// TIA Portal V17 export
// export: Created 2025-07-01T09:58:42.1462376Z, ExportSetting WithDefaults, DisplayName Totally Integrated Automation Portal, DisplayVersion V17 Update 8, DisplayName TIA Portal Openness, DisplayVersion V17 Update 8, DisplayName TIA Portal Version Control Interface, DisplayVersion V17, DisplayName SINAMICS Startdrive Advanced, DisplayVersion V17 SP2, DisplayName SINAMICS Startdrive G110M, G120, G120C, G120D, G120P, G115D, DisplayVersion V17 SP2, DisplayName SINAMICS Startdrive G130, G150, S120, S150, SINAMICS MV, S210, DisplayVersion V17 SP2, DisplayName STEP 7 Professional, DisplayVersion V17 Update 8, DisplayName SINUMERIK ONE STEP 7 Toolbox, DisplayVersion V17 Update 12, DisplayName SINUMERIK ONE PLC Basic Program Plus, DisplayVersion V17 Update 12, DisplayName SINUMERIK 840D sl STEP 7 Toolbox, DisplayVersion V17 Update 12, DisplayName STEP 7 Safety, DisplayVersion V17 Update 6, DisplayName WinCC Advanced, DisplayVersion V17 Update 8
FUNCTION "FC2034_DRY_CYCLE" : Void   // FC2034, LAD
{ S7_Optimized_Access := 'FALSE' }
AUTHOR : ETXETAR
VERSION : 1.0
// stored: AutoNumber false, IsIECCheckEnabled false, SetENOAutomatically false, UDAEnableTagReadback false
   VAR_TEMP
      O_BYTE_0 : Struct   // OPTIONS BYTE 0
         MANUAL_LOAD_WITH_LIFT : Bool;   // MANUAL LOAD WITH LIFTING DEVICE OPTION
      END_STRUCT;
      DISABLE_COMMAND : Bool;   // DRY CYCLE DISABLE COMMAND
   END_VAR
   VAR CONSTANT
      FC_NUMBER : DInt := 2034;
   END_VAR
   VAR_TEMP   // added for the SCL form of the ladder/FBD networks
      _w1 : Bool;
      _w2 : Bool;
   END_VAR
BEGIN

REGION Network 1: MANUAL LOAD WITH LIFTING DEVICE OPTION
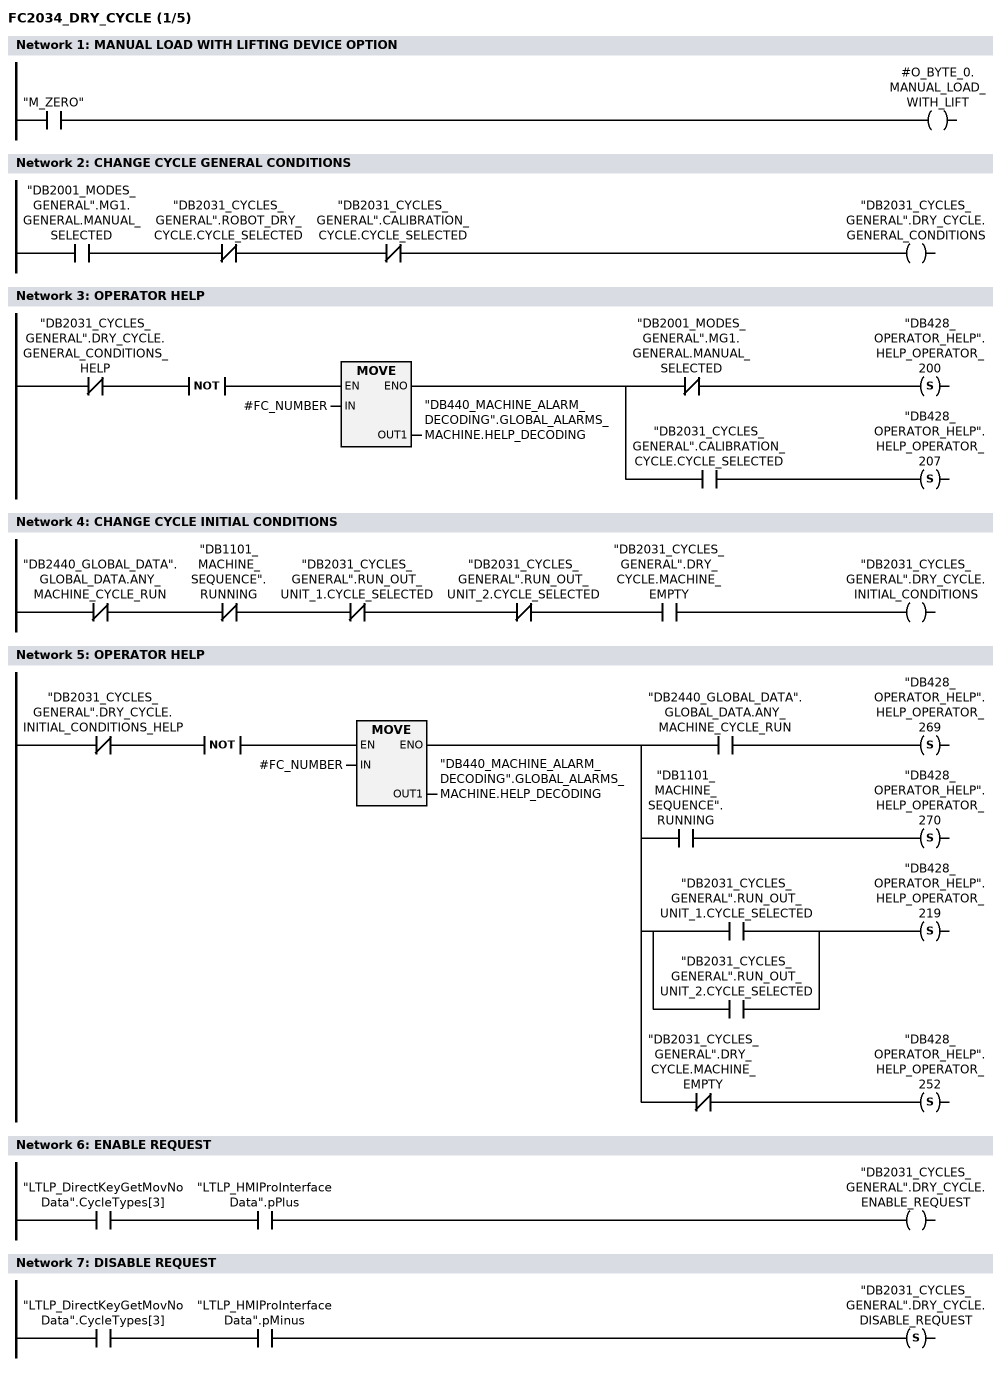
   RUNG wire#powerrail
      Contact( "M_ZERO" )
      Coil( #O_BYTE_0.MANUAL_LOAD_WITH_LIFT )
   END_RUNG
   // the same network as SCL:
   #O_BYTE_0.MANUAL_LOAD_WITH_LIFT := "M_ZERO";
END_REGION

REGION Network 2: CHANGE CYCLE GENERAL CONDITIONS
   RUNG wire#powerrail
      Contact( "DB2001_MODES_GENERAL".MG1.GENERAL.MANUAL_SELECTED )
      I_Contact( "DB2031_CYCLES_GENERAL".ROBOT_DRY_CYCLE.CYCLE_SELECTED )
      I_Contact( "DB2031_CYCLES_GENERAL".CALIBRATION_CYCLE.CYCLE_SELECTED )
      Coil( "DB2031_CYCLES_GENERAL".DRY_CYCLE.GENERAL_CONDITIONS )
   END_RUNG
   // the same network as SCL:
   "DB2031_CYCLES_GENERAL".DRY_CYCLE.GENERAL_CONDITIONS := "DB2001_MODES_GENERAL".MG1.GENERAL.MANUAL_SELECTED AND NOT "DB2031_CYCLES_GENERAL".ROBOT_DRY_CYCLE.CYCLE_SELECTED AND NOT "DB2031_CYCLES_GENERAL".CALIBRATION_CYCLE.CYCLE_SELECTED;
END_REGION

REGION Network 3: OPERATOR HELP
   RUNG wire#powerrail
      I_Contact( "DB2031_CYCLES_GENERAL".DRY_CYCLE.GENERAL_CONDITIONS_HELP )
      Not()
      { S7_GenerateENO := "TRUE" } Move(in := #FC_NUMBER, out1 => "DB440_MACHINE_ALARM_DECODING".GLOBAL_ALARMS_MACHINE.HELP_DECODING)
      wire#w1
      I_Contact( "DB2001_MODES_GENERAL".MG1.GENERAL.MANUAL_SELECTED )
      S_Coil( "DB428_OPERATOR_HELP".HELP_OPERATOR_200 )
   END_RUNG
   RUNG wire#w1
      Contact( "DB2031_CYCLES_GENERAL".CALIBRATION_CYCLE.CYCLE_SELECTED )
      S_Coil( "DB428_OPERATOR_HELP".HELP_OPERATOR_207 )
   END_RUNG
   // the same network as SCL:
   // ENO of a box is taken as its EN; it also drops when the box reports an error
   #_w1 := NOT (NOT "DB2031_CYCLES_GENERAL".DRY_CYCLE.GENERAL_CONDITIONS_HELP);
   IF #_w1 THEN "DB440_MACHINE_ALARM_DECODING".GLOBAL_ALARMS_MACHINE.HELP_DECODING := #FC_NUMBER; END_IF;
   IF #_w1 AND NOT "DB2001_MODES_GENERAL".MG1.GENERAL.MANUAL_SELECTED THEN
       "DB428_OPERATOR_HELP".HELP_OPERATOR_200 := TRUE;
   END_IF;
   IF #_w1 AND "DB2031_CYCLES_GENERAL".CALIBRATION_CYCLE.CYCLE_SELECTED THEN
       "DB428_OPERATOR_HELP".HELP_OPERATOR_207 := TRUE;
   END_IF;
END_REGION

REGION Network 4: CHANGE CYCLE INITIAL CONDITIONS
   RUNG wire#powerrail
      I_Contact( "DB2440_GLOBAL_DATA".GLOBAL_DATA.ANY_MACHINE_CYCLE_RUN )
      I_Contact( "DB1101_MACHINE_SEQUENCE".RUNNING )
      I_Contact( "DB2031_CYCLES_GENERAL".RUN_OUT_UNIT_1.CYCLE_SELECTED )
      I_Contact( "DB2031_CYCLES_GENERAL".RUN_OUT_UNIT_2.CYCLE_SELECTED )
      Contact( "DB2031_CYCLES_GENERAL".DRY_CYCLE.MACHINE_EMPTY )
      Coil( "DB2031_CYCLES_GENERAL".DRY_CYCLE.INITIAL_CONDITIONS )
   END_RUNG
   // the same network as SCL:
   "DB2031_CYCLES_GENERAL".DRY_CYCLE.INITIAL_CONDITIONS := NOT "DB2440_GLOBAL_DATA".GLOBAL_DATA.ANY_MACHINE_CYCLE_RUN AND NOT "DB1101_MACHINE_SEQUENCE".RUNNING AND NOT "DB2031_CYCLES_GENERAL".RUN_OUT_UNIT_1.CYCLE_SELECTED AND NOT "DB2031_CYCLES_GENERAL".RUN_OUT_UNIT_2.CYCLE_SELECTED AND "DB2031_CYCLES_GENERAL".DRY_CYCLE.MACHINE_EMPTY;
END_REGION

REGION Network 5: OPERATOR HELP
   RUNG wire#powerrail
      I_Contact( "DB2031_CYCLES_GENERAL".DRY_CYCLE.INITIAL_CONDITIONS_HELP )
      Not()
      { S7_GenerateENO := "TRUE" } Move(in := #FC_NUMBER, out1 => "DB440_MACHINE_ALARM_DECODING".GLOBAL_ALARMS_MACHINE.HELP_DECODING)
      wire#w1
      Contact( "DB2440_GLOBAL_DATA".GLOBAL_DATA.ANY_MACHINE_CYCLE_RUN )
      S_Coil( "DB428_OPERATOR_HELP".HELP_OPERATOR_269 )
   END_RUNG
   RUNG wire#w1
      Contact( "DB1101_MACHINE_SEQUENCE".RUNNING )
      S_Coil( "DB428_OPERATOR_HELP".HELP_OPERATOR_270 )
   END_RUNG
   RUNG wire#w1
      Contact( "DB2031_CYCLES_GENERAL".RUN_OUT_UNIT_1.CYCLE_SELECTED )
      wire#w2
      S_Coil( "DB428_OPERATOR_HELP".HELP_OPERATOR_219 )
   END_RUNG
   RUNG wire#w1
      Contact( "DB2031_CYCLES_GENERAL".RUN_OUT_UNIT_2.CYCLE_SELECTED )
   END_RUNG wire#w2
   RUNG wire#w1
      I_Contact( "DB2031_CYCLES_GENERAL".DRY_CYCLE.MACHINE_EMPTY )
      S_Coil( "DB428_OPERATOR_HELP".HELP_OPERATOR_252 )
   END_RUNG
   // the same network as SCL:
   // ENO of a box is taken as its EN; it also drops when the box reports an error
   #_w1 := NOT (NOT "DB2031_CYCLES_GENERAL".DRY_CYCLE.INITIAL_CONDITIONS_HELP);
   IF #_w1 THEN "DB440_MACHINE_ALARM_DECODING".GLOBAL_ALARMS_MACHINE.HELP_DECODING := #FC_NUMBER; END_IF;
   IF #_w1 AND "DB2440_GLOBAL_DATA".GLOBAL_DATA.ANY_MACHINE_CYCLE_RUN THEN
       "DB428_OPERATOR_HELP".HELP_OPERATOR_269 := TRUE;
   END_IF;
   IF #_w1 AND "DB1101_MACHINE_SEQUENCE".RUNNING THEN
       "DB428_OPERATOR_HELP".HELP_OPERATOR_270 := TRUE;
   END_IF;
   IF #_w1 AND ("DB2031_CYCLES_GENERAL".RUN_OUT_UNIT_1.CYCLE_SELECTED OR "DB2031_CYCLES_GENERAL".RUN_OUT_UNIT_2.CYCLE_SELECTED) THEN
       "DB428_OPERATOR_HELP".HELP_OPERATOR_219 := TRUE;
   END_IF;
   IF #_w1 AND NOT "DB2031_CYCLES_GENERAL".DRY_CYCLE.MACHINE_EMPTY THEN
       "DB428_OPERATOR_HELP".HELP_OPERATOR_252 := TRUE;
   END_IF;
END_REGION

REGION Network 6: ENABLE REQUEST
   RUNG wire#powerrail
      Contact( "LTLP_DirectKeyGetMovNoData".CycleTypes[3] )
      Contact( "LTLP_HMIProInterfaceData".pPlus )
      Coil( "DB2031_CYCLES_GENERAL".DRY_CYCLE.ENABLE_REQUEST )
   END_RUNG
   // the same network as SCL:
   "DB2031_CYCLES_GENERAL".DRY_CYCLE.ENABLE_REQUEST := "LTLP_DirectKeyGetMovNoData".CycleTypes[3] AND "LTLP_HMIProInterfaceData".pPlus;
END_REGION

REGION Network 7: DISABLE REQUEST
   RUNG wire#powerrail
      Contact( "LTLP_DirectKeyGetMovNoData".CycleTypes[3] )
      Contact( "LTLP_HMIProInterfaceData".pMinus )
      S_Coil( "DB2031_CYCLES_GENERAL".DRY_CYCLE.DISABLE_REQUEST )
   END_RUNG
   // the same network as SCL:
   IF "LTLP_DirectKeyGetMovNoData".CycleTypes[3] AND "LTLP_HMIProInterfaceData".pMinus THEN
       "DB2031_CYCLES_GENERAL".DRY_CYCLE.DISABLE_REQUEST := TRUE;
   END_IF;
END_REGION

REGION Network 8: ROBOT DRY CYCLE DISABLE COMMAND
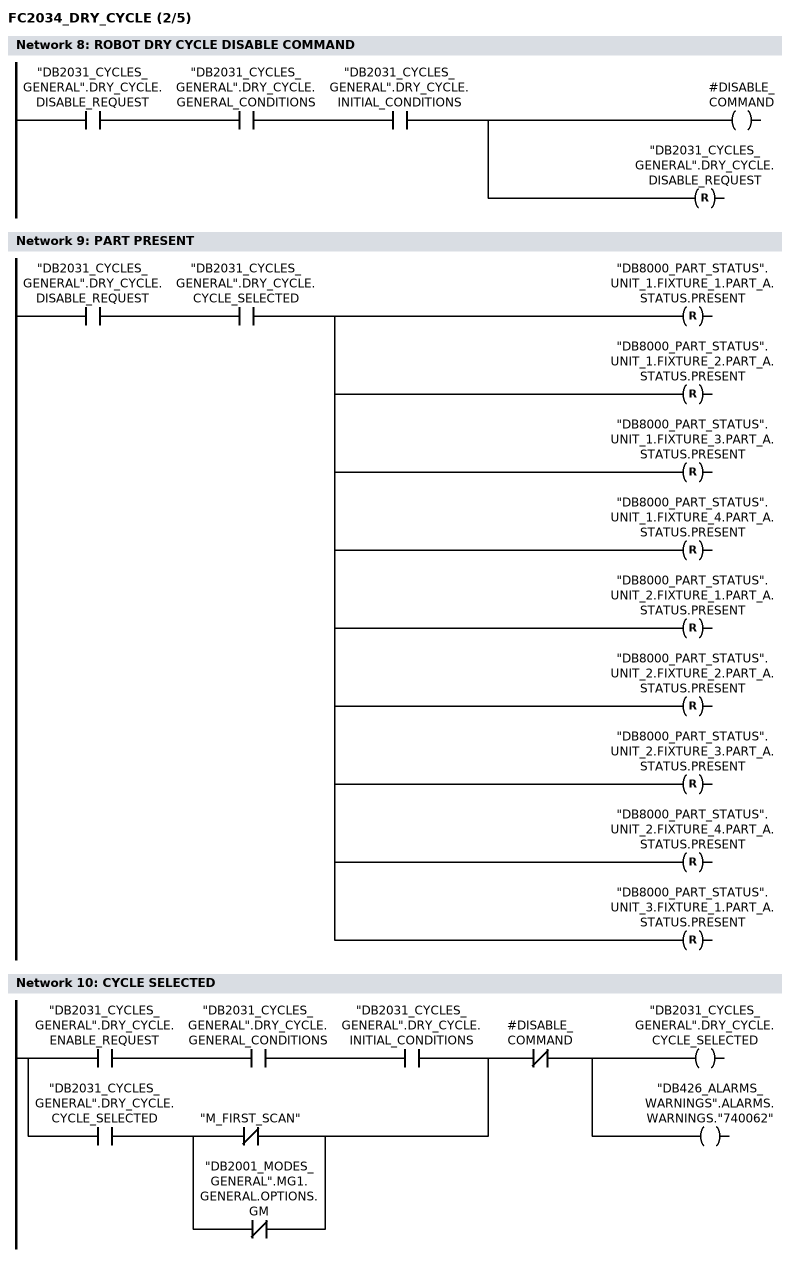
   RUNG wire#powerrail
      Contact( "DB2031_CYCLES_GENERAL".DRY_CYCLE.DISABLE_REQUEST )
      Contact( "DB2031_CYCLES_GENERAL".DRY_CYCLE.GENERAL_CONDITIONS )
      Contact( "DB2031_CYCLES_GENERAL".DRY_CYCLE.INITIAL_CONDITIONS )
      wire#w1
      Coil( #DISABLE_COMMAND )
   END_RUNG
   RUNG wire#w1
      R_Coil( "DB2031_CYCLES_GENERAL".DRY_CYCLE.DISABLE_REQUEST )
   END_RUNG
   // the same network as SCL:
   #DISABLE_COMMAND := "DB2031_CYCLES_GENERAL".DRY_CYCLE.DISABLE_REQUEST AND "DB2031_CYCLES_GENERAL".DRY_CYCLE.GENERAL_CONDITIONS AND "DB2031_CYCLES_GENERAL".DRY_CYCLE.INITIAL_CONDITIONS;
   IF #DISABLE_COMMAND THEN "DB2031_CYCLES_GENERAL".DRY_CYCLE.DISABLE_REQUEST := FALSE; END_IF;
END_REGION

REGION Network 9: PART PRESENT
   RUNG wire#powerrail
      Contact( "DB2031_CYCLES_GENERAL".DRY_CYCLE.DISABLE_REQUEST )
      Contact( "DB2031_CYCLES_GENERAL".DRY_CYCLE.CYCLE_SELECTED )
      wire#w1
      R_Coil( "DB8000_PART_STATUS".UNIT_1.FIXTURE_1.PART_A.STATUS.PRESENT )
   END_RUNG
   RUNG wire#w1
      R_Coil( "DB8000_PART_STATUS".UNIT_1.FIXTURE_2.PART_A.STATUS.PRESENT )
   END_RUNG
   RUNG wire#w1
      R_Coil( "DB8000_PART_STATUS".UNIT_1.FIXTURE_3.PART_A.STATUS.PRESENT )
   END_RUNG
   RUNG wire#w1
      R_Coil( "DB8000_PART_STATUS".UNIT_1.FIXTURE_4.PART_A.STATUS.PRESENT )
   END_RUNG
   RUNG wire#w1
      R_Coil( "DB8000_PART_STATUS".UNIT_2.FIXTURE_1.PART_A.STATUS.PRESENT )
   END_RUNG
   RUNG wire#w1
      R_Coil( "DB8000_PART_STATUS".UNIT_2.FIXTURE_2.PART_A.STATUS.PRESENT )
   END_RUNG
   RUNG wire#w1
      R_Coil( "DB8000_PART_STATUS".UNIT_2.FIXTURE_3.PART_A.STATUS.PRESENT )
   END_RUNG
   RUNG wire#w1
      R_Coil( "DB8000_PART_STATUS".UNIT_2.FIXTURE_4.PART_A.STATUS.PRESENT )
   END_RUNG
   RUNG wire#w1
      R_Coil( "DB8000_PART_STATUS".UNIT_3.FIXTURE_1.PART_A.STATUS.PRESENT )
   END_RUNG
   // the same network as SCL:
   IF "DB2031_CYCLES_GENERAL".DRY_CYCLE.DISABLE_REQUEST AND "DB2031_CYCLES_GENERAL".DRY_CYCLE.CYCLE_SELECTED THEN
       "DB8000_PART_STATUS".UNIT_1.FIXTURE_1.PART_A.STATUS.PRESENT := FALSE;
       "DB8000_PART_STATUS".UNIT_1.FIXTURE_2.PART_A.STATUS.PRESENT := FALSE;
       "DB8000_PART_STATUS".UNIT_1.FIXTURE_3.PART_A.STATUS.PRESENT := FALSE;
       "DB8000_PART_STATUS".UNIT_1.FIXTURE_4.PART_A.STATUS.PRESENT := FALSE;
       "DB8000_PART_STATUS".UNIT_2.FIXTURE_1.PART_A.STATUS.PRESENT := FALSE;
       "DB8000_PART_STATUS".UNIT_2.FIXTURE_2.PART_A.STATUS.PRESENT := FALSE;
       "DB8000_PART_STATUS".UNIT_2.FIXTURE_3.PART_A.STATUS.PRESENT := FALSE;
       "DB8000_PART_STATUS".UNIT_2.FIXTURE_4.PART_A.STATUS.PRESENT := FALSE;
       "DB8000_PART_STATUS".UNIT_3.FIXTURE_1.PART_A.STATUS.PRESENT := FALSE;
   END_IF;
END_REGION

REGION Network 10: CYCLE SELECTED
   RUNG wire#powerrail
      Contact( "DB2031_CYCLES_GENERAL".DRY_CYCLE.ENABLE_REQUEST )
      Contact( "DB2031_CYCLES_GENERAL".DRY_CYCLE.GENERAL_CONDITIONS )
      Contact( "DB2031_CYCLES_GENERAL".DRY_CYCLE.INITIAL_CONDITIONS )
      wire#w1
      I_Contact( #DISABLE_COMMAND )
      wire#w3
      Coil( "DB2031_CYCLES_GENERAL".DRY_CYCLE.CYCLE_SELECTED )
   END_RUNG
   RUNG wire#powerrail
      Contact( "DB2031_CYCLES_GENERAL".DRY_CYCLE.CYCLE_SELECTED )
      wire#w2
      I_Contact( "M_FIRST_SCAN" )
   END_RUNG wire#w1
   RUNG wire#w2
      I_Contact( "DB2001_MODES_GENERAL".MG1.GENERAL.OPTIONS.GM )
   END_RUNG wire#w1
   RUNG wire#w3
      Coil( "DB426_ALARMS_WARNINGS".ALARMS.WARNINGS."740062" )
   END_RUNG
   // the same network as SCL:
   "DB2031_CYCLES_GENERAL".DRY_CYCLE.CYCLE_SELECTED := (("DB2031_CYCLES_GENERAL".DRY_CYCLE.ENABLE_REQUEST AND "DB2031_CYCLES_GENERAL".DRY_CYCLE.GENERAL_CONDITIONS AND "DB2031_CYCLES_GENERAL".DRY_CYCLE.INITIAL_CONDITIONS) OR ("DB2031_CYCLES_GENERAL".DRY_CYCLE.CYCLE_SELECTED AND (NOT "M_FIRST_SCAN" OR NOT "DB2001_MODES_GENERAL".MG1.GENERAL.OPTIONS.GM))) AND NOT #DISABLE_COMMAND;
   "DB426_ALARMS_WARNINGS".ALARMS.WARNINGS."740062" := "DB2031_CYCLES_GENERAL".DRY_CYCLE.CYCLE_SELECTED;
END_REGION

REGION Network 11: WARNINGS
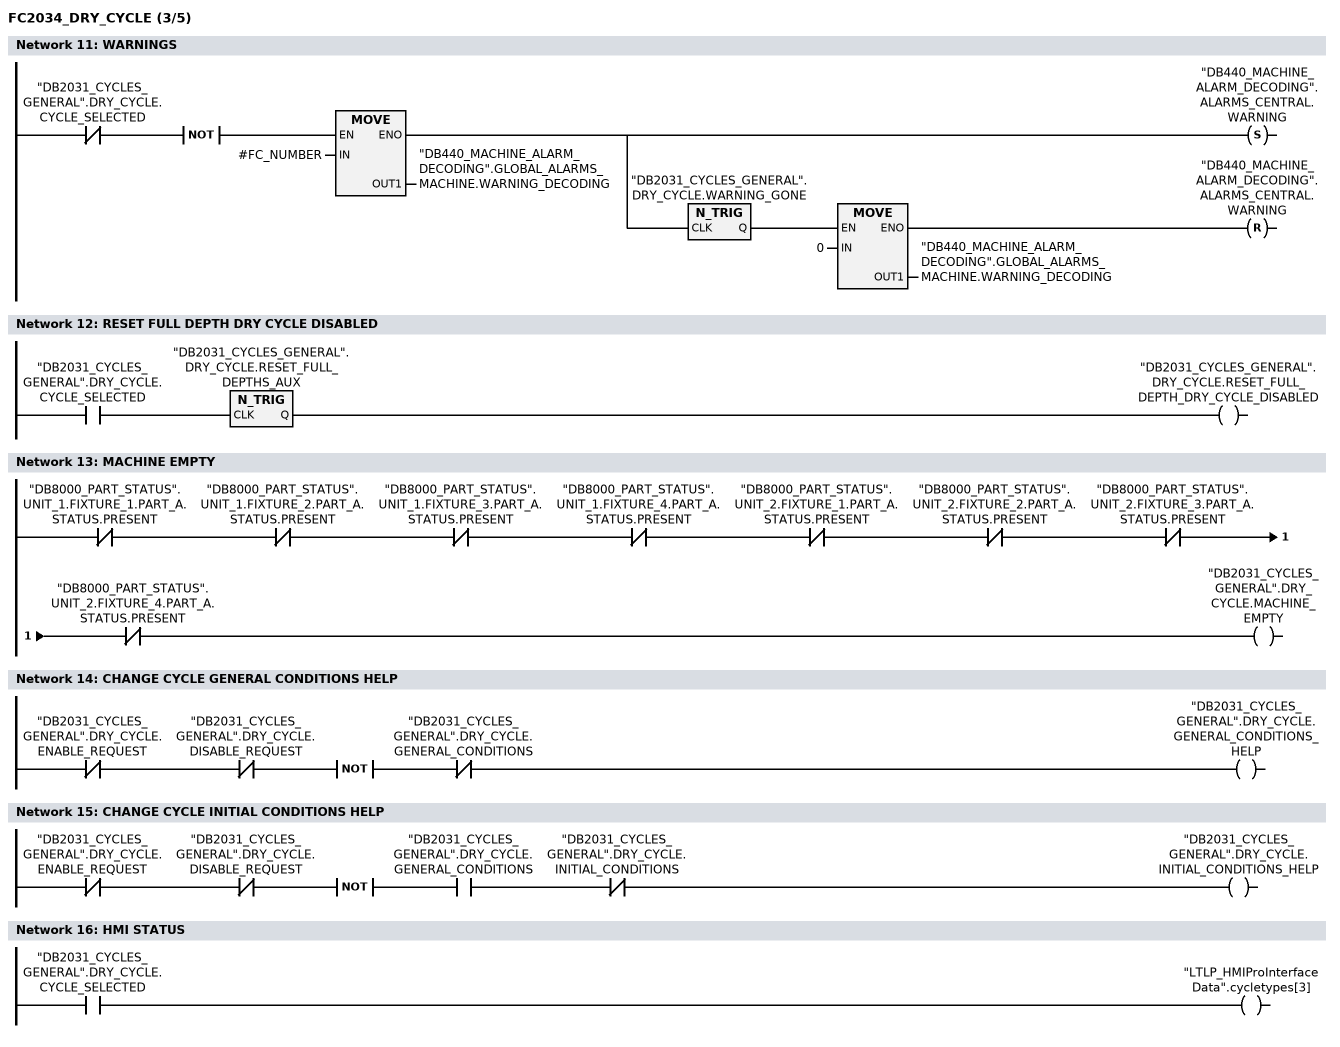
   RUNG wire#powerrail
      I_Contact( "DB2031_CYCLES_GENERAL".DRY_CYCLE.CYCLE_SELECTED )
      Not()
      Move(in := #FC_NUMBER, out1 => "DB440_MACHINE_ALARM_DECODING".GLOBAL_ALARMS_MACHINE.WARNING_DECODING)
      wire#w1
      S_Coil( "DB440_MACHINE_ALARM_DECODING".ALARMS_CENTRAL.WARNING )
   END_RUNG
   RUNG wire#w1
      N_Trig( "DB2031_CYCLES_GENERAL".DRY_CYCLE.WARNING_GONE )
      Move(in := 0, out1 => "DB440_MACHINE_ALARM_DECODING".GLOBAL_ALARMS_MACHINE.WARNING_DECODING)
      R_Coil( "DB440_MACHINE_ALARM_DECODING".ALARMS_CENTRAL.WARNING )
   END_RUNG
   // the same network as SCL:
   #_w1 := NOT (NOT "DB2031_CYCLES_GENERAL".DRY_CYCLE.CYCLE_SELECTED);
   IF #_w1 THEN
       "DB440_MACHINE_ALARM_DECODING".GLOBAL_ALARMS_MACHINE.WARNING_DECODING := #FC_NUMBER;
       "DB440_MACHINE_ALARM_DECODING".ALARMS_CENTRAL.WARNING := TRUE;
   END_IF;
   #_w2 := NOT #_w1 AND "DB2031_CYCLES_GENERAL".DRY_CYCLE.WARNING_GONE;   // falling edge
   "DB2031_CYCLES_GENERAL".DRY_CYCLE.WARNING_GONE := #_w1;
   IF #_w2 THEN
       "DB440_MACHINE_ALARM_DECODING".GLOBAL_ALARMS_MACHINE.WARNING_DECODING := 0;
       "DB440_MACHINE_ALARM_DECODING".ALARMS_CENTRAL.WARNING := FALSE;
   END_IF;
END_REGION

REGION Network 12: RESET FULL DEPTH DRY CYCLE DISABLED
   RUNG wire#powerrail
      Contact( "DB2031_CYCLES_GENERAL".DRY_CYCLE.CYCLE_SELECTED )
      N_Trig( "DB2031_CYCLES_GENERAL".DRY_CYCLE.RESET_FULL_DEPTHS_AUX )
      Coil( "DB2031_CYCLES_GENERAL".DRY_CYCLE.RESET_FULL_DEPTH_DRY_CYCLE_DISABLED )
   END_RUNG
   // the same network as SCL:
   #_w1 := NOT "DB2031_CYCLES_GENERAL".DRY_CYCLE.CYCLE_SELECTED AND "DB2031_CYCLES_GENERAL".DRY_CYCLE.RESET_FULL_DEPTHS_AUX;   // falling edge
   "DB2031_CYCLES_GENERAL".DRY_CYCLE.RESET_FULL_DEPTHS_AUX := "DB2031_CYCLES_GENERAL".DRY_CYCLE.CYCLE_SELECTED;
   "DB2031_CYCLES_GENERAL".DRY_CYCLE.RESET_FULL_DEPTH_DRY_CYCLE_DISABLED := #_w1;
END_REGION

REGION Network 13: MACHINE EMPTY
   RUNG wire#powerrail
      I_Contact( "DB8000_PART_STATUS".UNIT_1.FIXTURE_1.PART_A.STATUS.PRESENT )
      I_Contact( "DB8000_PART_STATUS".UNIT_1.FIXTURE_2.PART_A.STATUS.PRESENT )
      I_Contact( "DB8000_PART_STATUS".UNIT_1.FIXTURE_3.PART_A.STATUS.PRESENT )
      I_Contact( "DB8000_PART_STATUS".UNIT_1.FIXTURE_4.PART_A.STATUS.PRESENT )
      I_Contact( "DB8000_PART_STATUS".UNIT_2.FIXTURE_1.PART_A.STATUS.PRESENT )
      I_Contact( "DB8000_PART_STATUS".UNIT_2.FIXTURE_2.PART_A.STATUS.PRESENT )
      I_Contact( "DB8000_PART_STATUS".UNIT_2.FIXTURE_3.PART_A.STATUS.PRESENT )
      I_Contact( "DB8000_PART_STATUS".UNIT_2.FIXTURE_4.PART_A.STATUS.PRESENT )
      Coil( "DB2031_CYCLES_GENERAL".DRY_CYCLE.MACHINE_EMPTY )
   END_RUNG
   // the same network as SCL:
   "DB2031_CYCLES_GENERAL".DRY_CYCLE.MACHINE_EMPTY := NOT "DB8000_PART_STATUS".UNIT_1.FIXTURE_1.PART_A.STATUS.PRESENT AND NOT "DB8000_PART_STATUS".UNIT_1.FIXTURE_2.PART_A.STATUS.PRESENT AND NOT "DB8000_PART_STATUS".UNIT_1.FIXTURE_3.PART_A.STATUS.PRESENT AND NOT "DB8000_PART_STATUS".UNIT_1.FIXTURE_4.PART_A.STATUS.PRESENT AND NOT "DB8000_PART_STATUS".UNIT_2.FIXTURE_1.PART_A.STATUS.PRESENT AND NOT "DB8000_PART_STATUS".UNIT_2.FIXTURE_2.PART_A.STATUS.PRESENT AND NOT "DB8000_PART_STATUS".UNIT_2.FIXTURE_3.PART_A.STATUS.PRESENT AND NOT "DB8000_PART_STATUS".UNIT_2.FIXTURE_4.PART_A.STATUS.PRESENT;
END_REGION

REGION Network 14: CHANGE CYCLE GENERAL CONDITIONS HELP
   RUNG wire#powerrail
      I_Contact( "DB2031_CYCLES_GENERAL".DRY_CYCLE.ENABLE_REQUEST )
      I_Contact( "DB2031_CYCLES_GENERAL".DRY_CYCLE.DISABLE_REQUEST )
      Not()
      I_Contact( "DB2031_CYCLES_GENERAL".DRY_CYCLE.GENERAL_CONDITIONS )
      Coil( "DB2031_CYCLES_GENERAL".DRY_CYCLE.GENERAL_CONDITIONS_HELP )
   END_RUNG
   // the same network as SCL:
   "DB2031_CYCLES_GENERAL".DRY_CYCLE.GENERAL_CONDITIONS_HELP := NOT (NOT "DB2031_CYCLES_GENERAL".DRY_CYCLE.ENABLE_REQUEST AND NOT "DB2031_CYCLES_GENERAL".DRY_CYCLE.DISABLE_REQUEST) AND NOT "DB2031_CYCLES_GENERAL".DRY_CYCLE.GENERAL_CONDITIONS;
END_REGION

REGION Network 15: CHANGE CYCLE INITIAL CONDITIONS HELP
   RUNG wire#powerrail
      I_Contact( "DB2031_CYCLES_GENERAL".DRY_CYCLE.ENABLE_REQUEST )
      I_Contact( "DB2031_CYCLES_GENERAL".DRY_CYCLE.DISABLE_REQUEST )
      Not()
      Contact( "DB2031_CYCLES_GENERAL".DRY_CYCLE.GENERAL_CONDITIONS )
      I_Contact( "DB2031_CYCLES_GENERAL".DRY_CYCLE.INITIAL_CONDITIONS )
      Coil( "DB2031_CYCLES_GENERAL".DRY_CYCLE.INITIAL_CONDITIONS_HELP )
   END_RUNG
   // the same network as SCL:
   "DB2031_CYCLES_GENERAL".DRY_CYCLE.INITIAL_CONDITIONS_HELP := NOT (NOT "DB2031_CYCLES_GENERAL".DRY_CYCLE.ENABLE_REQUEST AND NOT "DB2031_CYCLES_GENERAL".DRY_CYCLE.DISABLE_REQUEST) AND "DB2031_CYCLES_GENERAL".DRY_CYCLE.GENERAL_CONDITIONS AND NOT "DB2031_CYCLES_GENERAL".DRY_CYCLE.INITIAL_CONDITIONS;
END_REGION

REGION Network 16: HMI STATUS
   RUNG wire#powerrail
      Contact( "DB2031_CYCLES_GENERAL".DRY_CYCLE.CYCLE_SELECTED )
      Coil( "LTLP_HMIProInterfaceData".cycletypes[3] )
   END_RUNG
   // the same network as SCL:
   "LTLP_HMIProInterfaceData".cycletypes[3] := "DB2031_CYCLES_GENERAL".DRY_CYCLE.CYCLE_SELECTED;
END_REGION

REGION Network 17: UNIT 01 VIRTUAL PART PRESENT
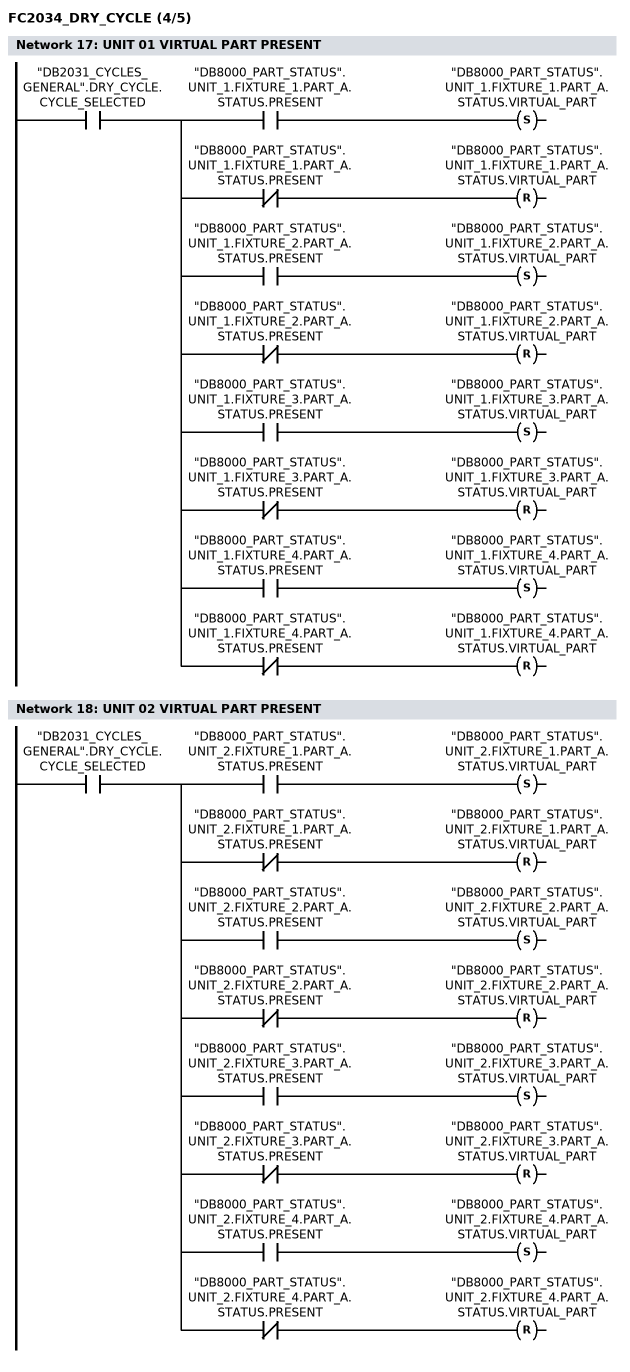
   RUNG wire#powerrail
      Contact( "DB2031_CYCLES_GENERAL".DRY_CYCLE.CYCLE_SELECTED )
      wire#w1
      Contact( "DB8000_PART_STATUS".UNIT_1.FIXTURE_1.PART_A.STATUS.PRESENT )
      S_Coil( "DB8000_PART_STATUS".UNIT_1.FIXTURE_1.PART_A.STATUS.VIRTUAL_PART )
   END_RUNG
   RUNG wire#w1
      I_Contact( "DB8000_PART_STATUS".UNIT_1.FIXTURE_1.PART_A.STATUS.PRESENT )
      R_Coil( "DB8000_PART_STATUS".UNIT_1.FIXTURE_1.PART_A.STATUS.VIRTUAL_PART )
   END_RUNG
   RUNG wire#w1
      Contact( "DB8000_PART_STATUS".UNIT_1.FIXTURE_2.PART_A.STATUS.PRESENT )
      S_Coil( "DB8000_PART_STATUS".UNIT_1.FIXTURE_2.PART_A.STATUS.VIRTUAL_PART )
   END_RUNG
   RUNG wire#w1
      I_Contact( "DB8000_PART_STATUS".UNIT_1.FIXTURE_2.PART_A.STATUS.PRESENT )
      R_Coil( "DB8000_PART_STATUS".UNIT_1.FIXTURE_2.PART_A.STATUS.VIRTUAL_PART )
   END_RUNG
   RUNG wire#w1
      Contact( "DB8000_PART_STATUS".UNIT_1.FIXTURE_3.PART_A.STATUS.PRESENT )
      S_Coil( "DB8000_PART_STATUS".UNIT_1.FIXTURE_3.PART_A.STATUS.VIRTUAL_PART )
   END_RUNG
   RUNG wire#w1
      I_Contact( "DB8000_PART_STATUS".UNIT_1.FIXTURE_3.PART_A.STATUS.PRESENT )
      R_Coil( "DB8000_PART_STATUS".UNIT_1.FIXTURE_3.PART_A.STATUS.VIRTUAL_PART )
   END_RUNG
   RUNG wire#w1
      Contact( "DB8000_PART_STATUS".UNIT_1.FIXTURE_4.PART_A.STATUS.PRESENT )
      S_Coil( "DB8000_PART_STATUS".UNIT_1.FIXTURE_4.PART_A.STATUS.VIRTUAL_PART )
   END_RUNG
   RUNG wire#w1
      I_Contact( "DB8000_PART_STATUS".UNIT_1.FIXTURE_4.PART_A.STATUS.PRESENT )
      R_Coil( "DB8000_PART_STATUS".UNIT_1.FIXTURE_4.PART_A.STATUS.VIRTUAL_PART )
   END_RUNG
   // the same network as SCL:
   IF "DB2031_CYCLES_GENERAL".DRY_CYCLE.CYCLE_SELECTED AND "DB8000_PART_STATUS".UNIT_1.FIXTURE_1.PART_A.STATUS.PRESENT THEN
       "DB8000_PART_STATUS".UNIT_1.FIXTURE_1.PART_A.STATUS.VIRTUAL_PART := TRUE;
   END_IF;
   IF "DB2031_CYCLES_GENERAL".DRY_CYCLE.CYCLE_SELECTED AND NOT "DB8000_PART_STATUS".UNIT_1.FIXTURE_1.PART_A.STATUS.PRESENT THEN
       "DB8000_PART_STATUS".UNIT_1.FIXTURE_1.PART_A.STATUS.VIRTUAL_PART := FALSE;
   END_IF;
   IF "DB2031_CYCLES_GENERAL".DRY_CYCLE.CYCLE_SELECTED AND "DB8000_PART_STATUS".UNIT_1.FIXTURE_2.PART_A.STATUS.PRESENT THEN
       "DB8000_PART_STATUS".UNIT_1.FIXTURE_2.PART_A.STATUS.VIRTUAL_PART := TRUE;
   END_IF;
   IF "DB2031_CYCLES_GENERAL".DRY_CYCLE.CYCLE_SELECTED AND NOT "DB8000_PART_STATUS".UNIT_1.FIXTURE_2.PART_A.STATUS.PRESENT THEN
       "DB8000_PART_STATUS".UNIT_1.FIXTURE_2.PART_A.STATUS.VIRTUAL_PART := FALSE;
   END_IF;
   IF "DB2031_CYCLES_GENERAL".DRY_CYCLE.CYCLE_SELECTED AND "DB8000_PART_STATUS".UNIT_1.FIXTURE_3.PART_A.STATUS.PRESENT THEN
       "DB8000_PART_STATUS".UNIT_1.FIXTURE_3.PART_A.STATUS.VIRTUAL_PART := TRUE;
   END_IF;
   IF "DB2031_CYCLES_GENERAL".DRY_CYCLE.CYCLE_SELECTED AND NOT "DB8000_PART_STATUS".UNIT_1.FIXTURE_3.PART_A.STATUS.PRESENT THEN
       "DB8000_PART_STATUS".UNIT_1.FIXTURE_3.PART_A.STATUS.VIRTUAL_PART := FALSE;
   END_IF;
   IF "DB2031_CYCLES_GENERAL".DRY_CYCLE.CYCLE_SELECTED AND "DB8000_PART_STATUS".UNIT_1.FIXTURE_4.PART_A.STATUS.PRESENT THEN
       "DB8000_PART_STATUS".UNIT_1.FIXTURE_4.PART_A.STATUS.VIRTUAL_PART := TRUE;
   END_IF;
   IF "DB2031_CYCLES_GENERAL".DRY_CYCLE.CYCLE_SELECTED AND NOT "DB8000_PART_STATUS".UNIT_1.FIXTURE_4.PART_A.STATUS.PRESENT THEN
       "DB8000_PART_STATUS".UNIT_1.FIXTURE_4.PART_A.STATUS.VIRTUAL_PART := FALSE;
   END_IF;
END_REGION

REGION Network 18: UNIT 02 VIRTUAL PART PRESENT
   RUNG wire#powerrail
      Contact( "DB2031_CYCLES_GENERAL".DRY_CYCLE.CYCLE_SELECTED )
      wire#w1
      Contact( "DB8000_PART_STATUS".UNIT_2.FIXTURE_1.PART_A.STATUS.PRESENT )
      S_Coil( "DB8000_PART_STATUS".UNIT_2.FIXTURE_1.PART_A.STATUS.VIRTUAL_PART )
   END_RUNG
   RUNG wire#w1
      I_Contact( "DB8000_PART_STATUS".UNIT_2.FIXTURE_1.PART_A.STATUS.PRESENT )
      R_Coil( "DB8000_PART_STATUS".UNIT_2.FIXTURE_1.PART_A.STATUS.VIRTUAL_PART )
   END_RUNG
   RUNG wire#w1
      Contact( "DB8000_PART_STATUS".UNIT_2.FIXTURE_2.PART_A.STATUS.PRESENT )
      S_Coil( "DB8000_PART_STATUS".UNIT_2.FIXTURE_2.PART_A.STATUS.VIRTUAL_PART )
   END_RUNG
   RUNG wire#w1
      I_Contact( "DB8000_PART_STATUS".UNIT_2.FIXTURE_2.PART_A.STATUS.PRESENT )
      R_Coil( "DB8000_PART_STATUS".UNIT_2.FIXTURE_2.PART_A.STATUS.VIRTUAL_PART )
   END_RUNG
   RUNG wire#w1
      Contact( "DB8000_PART_STATUS".UNIT_2.FIXTURE_3.PART_A.STATUS.PRESENT )
      S_Coil( "DB8000_PART_STATUS".UNIT_2.FIXTURE_3.PART_A.STATUS.VIRTUAL_PART )
   END_RUNG
   RUNG wire#w1
      I_Contact( "DB8000_PART_STATUS".UNIT_2.FIXTURE_3.PART_A.STATUS.PRESENT )
      R_Coil( "DB8000_PART_STATUS".UNIT_2.FIXTURE_3.PART_A.STATUS.VIRTUAL_PART )
   END_RUNG
   RUNG wire#w1
      Contact( "DB8000_PART_STATUS".UNIT_2.FIXTURE_4.PART_A.STATUS.PRESENT )
      S_Coil( "DB8000_PART_STATUS".UNIT_2.FIXTURE_4.PART_A.STATUS.VIRTUAL_PART )
   END_RUNG
   RUNG wire#w1
      I_Contact( "DB8000_PART_STATUS".UNIT_2.FIXTURE_4.PART_A.STATUS.PRESENT )
      R_Coil( "DB8000_PART_STATUS".UNIT_2.FIXTURE_4.PART_A.STATUS.VIRTUAL_PART )
   END_RUNG
   // the same network as SCL:
   IF "DB2031_CYCLES_GENERAL".DRY_CYCLE.CYCLE_SELECTED AND "DB8000_PART_STATUS".UNIT_2.FIXTURE_1.PART_A.STATUS.PRESENT THEN
       "DB8000_PART_STATUS".UNIT_2.FIXTURE_1.PART_A.STATUS.VIRTUAL_PART := TRUE;
   END_IF;
   IF "DB2031_CYCLES_GENERAL".DRY_CYCLE.CYCLE_SELECTED AND NOT "DB8000_PART_STATUS".UNIT_2.FIXTURE_1.PART_A.STATUS.PRESENT THEN
       "DB8000_PART_STATUS".UNIT_2.FIXTURE_1.PART_A.STATUS.VIRTUAL_PART := FALSE;
   END_IF;
   IF "DB2031_CYCLES_GENERAL".DRY_CYCLE.CYCLE_SELECTED AND "DB8000_PART_STATUS".UNIT_2.FIXTURE_2.PART_A.STATUS.PRESENT THEN
       "DB8000_PART_STATUS".UNIT_2.FIXTURE_2.PART_A.STATUS.VIRTUAL_PART := TRUE;
   END_IF;
   IF "DB2031_CYCLES_GENERAL".DRY_CYCLE.CYCLE_SELECTED AND NOT "DB8000_PART_STATUS".UNIT_2.FIXTURE_2.PART_A.STATUS.PRESENT THEN
       "DB8000_PART_STATUS".UNIT_2.FIXTURE_2.PART_A.STATUS.VIRTUAL_PART := FALSE;
   END_IF;
   IF "DB2031_CYCLES_GENERAL".DRY_CYCLE.CYCLE_SELECTED AND "DB8000_PART_STATUS".UNIT_2.FIXTURE_3.PART_A.STATUS.PRESENT THEN
       "DB8000_PART_STATUS".UNIT_2.FIXTURE_3.PART_A.STATUS.VIRTUAL_PART := TRUE;
   END_IF;
   IF "DB2031_CYCLES_GENERAL".DRY_CYCLE.CYCLE_SELECTED AND NOT "DB8000_PART_STATUS".UNIT_2.FIXTURE_3.PART_A.STATUS.PRESENT THEN
       "DB8000_PART_STATUS".UNIT_2.FIXTURE_3.PART_A.STATUS.VIRTUAL_PART := FALSE;
   END_IF;
   IF "DB2031_CYCLES_GENERAL".DRY_CYCLE.CYCLE_SELECTED AND "DB8000_PART_STATUS".UNIT_2.FIXTURE_4.PART_A.STATUS.PRESENT THEN
       "DB8000_PART_STATUS".UNIT_2.FIXTURE_4.PART_A.STATUS.VIRTUAL_PART := TRUE;
   END_IF;
   IF "DB2031_CYCLES_GENERAL".DRY_CYCLE.CYCLE_SELECTED AND NOT "DB8000_PART_STATUS".UNIT_2.FIXTURE_4.PART_A.STATUS.PRESENT THEN
       "DB8000_PART_STATUS".UNIT_2.FIXTURE_4.PART_A.STATUS.VIRTUAL_PART := FALSE;
   END_IF;
END_REGION

REGION Network 19: UNIT 03 VIRTUAL PART PRESENT
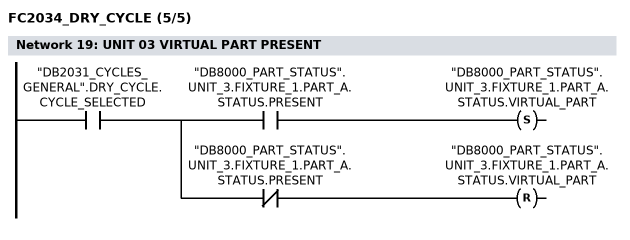
   RUNG wire#powerrail
      Contact( "DB2031_CYCLES_GENERAL".DRY_CYCLE.CYCLE_SELECTED )
      wire#w1
      Contact( "DB8000_PART_STATUS".UNIT_3.FIXTURE_1.PART_A.STATUS.PRESENT )
      S_Coil( "DB8000_PART_STATUS".UNIT_3.FIXTURE_1.PART_A.STATUS.VIRTUAL_PART )
   END_RUNG
   RUNG wire#w1
      I_Contact( "DB8000_PART_STATUS".UNIT_3.FIXTURE_1.PART_A.STATUS.PRESENT )
      R_Coil( "DB8000_PART_STATUS".UNIT_3.FIXTURE_1.PART_A.STATUS.VIRTUAL_PART )
   END_RUNG
   // the same network as SCL:
   IF "DB2031_CYCLES_GENERAL".DRY_CYCLE.CYCLE_SELECTED AND "DB8000_PART_STATUS".UNIT_3.FIXTURE_1.PART_A.STATUS.PRESENT THEN
       "DB8000_PART_STATUS".UNIT_3.FIXTURE_1.PART_A.STATUS.VIRTUAL_PART := TRUE;
   END_IF;
   IF "DB2031_CYCLES_GENERAL".DRY_CYCLE.CYCLE_SELECTED AND NOT "DB8000_PART_STATUS".UNIT_3.FIXTURE_1.PART_A.STATUS.PRESENT THEN
       "DB8000_PART_STATUS".UNIT_3.FIXTURE_1.PART_A.STATUS.VIRTUAL_PART := FALSE;
   END_IF;
END_REGION
END_FUNCTION
